// TIA Portal V15.1 export
// export: Created 2026-01-09T13:45:11.6525328Z, ExportSetting WithDefaults, WithReadOnly, DisplayName Totally Integrated Automation Portal, DisplayVersion V15.1 Update 8, DisplayName TIA Portal Openness, DisplayVersion V15.1 Update 8, DisplayName STEP 7 Professional, DisplayVersion V15.1 Update 8, DisplayName WinCC Advanced, DisplayVersion V15.1 Update 8
DATA_BLOCK "C#4_WD_WEIGHT"   // DB4
{ S7_Optimized_Access := 'FALSE' }
VERSION : 0.1
// stored: AutoNumber true, CodeModifiedDate 2024-09-25T16:02:28.9173662Z, CompileDate 2025-08-30T17:40:33.07032Z, CreationDate 2024-10-12T12:36:08.0193576Z, DBAccessibleFromOPCUA true, InterfaceModifiedDate 2024-09-25T16:02:28.9173662Z, IsConsistent true, IsKnowHowProtected false, IsOnlyStoredInLoadMemory false, IsPLCDB false, IsWriteProtectedInAS false, ModifiedDate 2024-10-13T07:08:48.1421634Z, ParameterModified 2024-09-25T16:02:28.9173662Z, StructureModified 2024-09-25T16:02:28.9173662Z
   VAR RETAIN
      "W_AG1_TG.DLC" : Real;   // Phễu cân Cốt liệu 1_Thời gian trễ cân
      "W_AG1_TG.DLX" : Real;   // Phễu cân Cốt liệu 1_Thời gian trễ xả
      "W_AG1_TG.DLD" : Real;   // Phễu cân Cốt liệu 1_Thời gian trễ đóng cân
      "W_AG1_KL.BRO" : Real;   // Phễu cân Cốt liệu 1_Khối lượng báo rỗng
      "W_AG1_KL.RUG" : Real;   // Phễu cân Cốt liệu 1_Khối lượng rung cân
      "W_AG1_TG.ON_RUNG" : Real;   // Phễu cân Cốt liệu 1_Thời gian bật rung
      "W_AG1_TG.OF_RUNG" : Real;   // Phễu cân Cốt liệu 1_Thời gian tắt rung
      "W_FD1_TG.DLC" : Real;   // Phễu cân FD 1_Thời gian trễ cân
      "W_FD1_TG.DLX" : Real;   // Phễu cân FD 1_Thời gian trễ xả
      "W_FD1_TG.DLD" : Real;   // Phễu cân FD 1_Thời gian trễ đóng cân
      "W_FD1_KL.BRO" : Real;   // Phễu cân FD 1_Khối lượng báo rỗng
      "W_FD1_KL.RUG" : Real;   // Phễu cân FD1_Khối lượng rung cân
      "W_FD1_TG.ON_RUNG" : Real;   // Phễu cân FD 1_Thời gian bật rung
      "W_FD1_TG.OF_RUNG" : Real;   // Phễu cân FD 1_Thời gian tắt rung
      "W_AP1_TG.DLC" : Real;   // Phễu cân Nhựa 1_Thời gian trễ cân
      "W_AP1_TG.DLX" : Real;   // Phễu cân Nhựa 1_Thời gian trễ xả
      "W_AP1_TG.DLD" : Real;   // Phễu cân Nhựa 1_Thời gian trễ đóng cân
      "W_AP1_KL.BRO" : Real;   // Phễu cân Nhựa 1_Khối lượng báo rỗng
      "W_SB1_TG.DLC" : Real;   // Phễu cân SBS 1_Thời gian trễ cân
      "W_SB1_TG.DLX" : Real;   // Phễu cân SBS 1_Thời gian trễ xả
      "W_SB1_TG.DLD" { ExternalWritable := 'False'} : Real;   // Phễu cân SBS 1_Thời gian trễ đóng cân
      "W_SB1_KL.BRO" : Real;   // Phễu cân SBS 1_Khối lượng báo rỗng
      "W_SB1_KL.RUG" : Real;   // Phễu cân SBS 1_Khối lượng rung cân
      "W_SB1_TG.ON_RUNG" : Real;   // Phễu cân SBS 1_Thời gian bật rung
      "W_SB1_TG.OF_RUNG" : Real;   // Phễu cân SBS 1_Thời gian tắt rung
      SO_ME_TRON : Real;   // Số mẻ cần trộn
      SV_AG1 : Real;   // Khối lượng Cần cân Cốt liệu 1
      SV_AG2 : Real;   // Khối lượng Cần cân Cốt liệu 2
      SV_AG3 : Real;   // Khối lượng Cần cân Cốt liệu 3
      SV_AG4 : Real;   // Khối lượng Cần cân Cốt liệu 4
      SV_AG5 : Real;   // Khối lượng Cần cân Cốt liệu 5
      SV_FD1 : Real;   // Khối lượng Cần cân FD 1
      SV_AP1 : Real;   // Khối lượng Cần cân Nhựa 1
      SV_SB1 : Real;   // Khối lượng Cần cân SBS 1
   END_VAR
BEGIN
END_DATA_BLOCK
